FUNCTION_BLOCK FB_DynamicMatrix_Test EXTENDS FB_TestSuite
VAR_INPUT
END_VAR
VAR_OUTPUT
END_VAR
VAR
END_VAR

WhenDeclaredExpectNoMemoryAllocated();
WhenInitiallyResizedExpectMemoryAllocated();
WhenResizedBiggerExpectMoreMemoryAllocated();
WhenResizedSmallerExpectLessMemoryAllocated();
WhenResizedToZeroExpectNoMemoryAllocated();

METHOD PRIVATE WhenDeclaredExpectNoMemoryAllocated
VAR_INPUT
END_VAR
VAR
	M : DynamicMatrix;
	
	ExpectedBufferSize : ULINT := 0;
	ExpectedBufferCount : ULINT := 0;
	
	ActualBufferSize : ULINT;
	ActualBufferCount : ULINT;
END_VAR
TEST('WhenDeclaredExpectNoMemoryAllocated');

// @TEST-RUN
ActualBufferSize := M.MemManager.nAllocatedSize;
ActualBufferCount := M.MemManager.nBufferCount;

// @TEST-ASSERT
AssertEquals(Expected := ExpectedBufferSize,
	Actual := ActualBufferSize,
	Message := 'Matrix buffer size not correct');
AssertEquals(Expected := ExpectedBufferCount,
	Actual := ActualBufferCount,
	Message := 'Matrix buffer count not correct');
	
TEST_FINISHED();
END_METHOD

METHOD PRIVATE WhenInitiallyResizedExpectMemoryAllocated
VAR_INPUT
END_VAR

VAR
	M : DynamicMatrix;
	ResizeSuccess : BOOL;
	
	ExpectedBufferSize : ULINT := 1*SIZEOF(LREAL) + SIZEOF(ULINT);
	ExpectedBufferCount : ULINT := 1;
	
	ActualBufferSize : ULINT;
	ActualBufferCount : ULINT;
END_VAR
TEST('WhenInitiallyResizedExpectMemoryAllocated');

// @TEST-RUN
ResizeSuccess := M.Resize(1,1,FALSE,TRUE);

ActualBufferSize := M.MemManager.nAllocatedSize;
ActualBufferCount := M.MemManager.nBufferCount;


// @TEST-ASSERT
AssertTrue(Condition :=ResizeSuccess,
	message := 'Error on valid initial resize');
AssertEquals(Expected := ExpectedBufferSize,
	Actual := ActualBufferSize,
	Message := 'Matrix buffer size not correct');
AssertEquals(Expected := ExpectedBufferCount,
	Actual := ActualBufferCount,
	Message := 'Matrix buffer count not correct');
	
TEST_FINISHED();
END_METHOD

METHOD PRIVATE WhenResizedBiggerExpectMoreMemoryAllocated
VAR_INPUT
END_VAR
VAR
	M : DynamicMatrix;
	InitialResizeSuccess : BOOL;
	SecondResizeSuccess : BOOL;
	
	ExpectedBufferSize : ULINT := 4*SIZEOF(LREAL) + SIZEOF(ULINT);
	ExpectedBufferCount : ULINT := 1;
	
	ActualBufferSize : ULINT;
	ActualBufferCount : ULINT;
END_VAR
TEST('WhenResizedBiggerExpectMoreMemoryAllocated');

// @TEST-RUN
InitialResizeSuccess := M.Resize(1,1,FALSE,TRUE);
SecondResizeSuccess := M.Resize(2,2,FALSE,TRUE);

ActualBufferSize := M.MemManager.nAllocatedSize;
ActualBufferCount := M.MemManager.nBufferCount;

// @TEST-ASSERT
AssertTrue(Condition :=InitialResizeSuccess,
	message := 'Error on valid initial resize');
AssertTrue(Condition :=SecondResizeSuccess,
	message := 'Error on valid second resize');
AssertEquals(Expected := ExpectedBufferSize,
	Actual := ActualBufferSize,
	Message := 'Matrix buffer size not correct');
AssertEquals(Expected := ExpectedBufferCount,
	Actual := ActualBufferCount,
	Message := 'Matrix buffer count not correct');
	
TEST_FINISHED();
END_METHOD

METHOD PRIVATE WhenResizedSmallerExpectLessMemoryAllocated
VAR_INPUT
END_VAR
VAR
	M : DynamicMatrix;
	InitialResizeSuccess : BOOL;
	SecondResizeSuccess : BOOL;
	
	ExpectedBufferSize : ULINT := 1*SIZEOF(LREAL) + SIZEOF(ULINT);
	ExpectedBufferCount : ULINT := 1;
	
	ActualBufferSize : ULINT;
	ActualBufferCount : ULINT;
END_VAR
TEST('WhenResizedSmallerExpectLessMemoryAllocated');

// @TEST-RUN
InitialResizeSuccess := M.Resize(2,2,FALSE,TRUE);
SecondResizeSuccess := M.Resize(1,1,FALSE,TRUE);

ActualBufferSize := M.MemManager.nAllocatedSize;
ActualBufferCount := M.MemManager.nBufferCount;

// @TEST-ASSERT
AssertTrue(Condition :=InitialResizeSuccess,
	message := 'Error on valid initial resize');
AssertTrue(Condition :=SecondResizeSuccess,
	message := 'Error on valid second resize');
AssertEquals(Expected := ExpectedBufferSize,
	Actual := ActualBufferSize,
	Message := 'Matrix buffer size not correct');
AssertEquals(Expected := ExpectedBufferCount,
	Actual := ActualBufferCount,
	Message := 'Matrix buffer count not correct');
	
TEST_FINISHED();
END_METHOD

METHOD PRIVATE WhenResizedToZeroExpectNoMemoryAllocated
VAR_INPUT
END_VAR
VAR
	M : DynamicMatrix;
	InitialResizeSuccess : BOOL;
	SecondResizeSuccess : BOOL;
	
	ExpectedBufferSize : ULINT := 0;
	ExpectedBufferCount : ULINT := 0;
	
	ActualBufferSize : ULINT;
	ActualBufferCount : ULINT;
END_VAR
TEST('WhenResizedToZeroExpectNoMemoryAllocated');

// @TEST-RUN
InitialResizeSuccess := M.Resize(1,1,FALSE,TRUE);
SecondResizeSuccess := M.Resize(0,0,FALSE,TRUE);

ActualBufferSize := M.MemManager.nAllocatedSize;
ActualBufferCount := M.MemManager.nBufferCount;

// @TEST-ASSERT
AssertTrue(Condition :=InitialResizeSuccess,
	message := 'Error on valid initial resize');
AssertTrue(Condition :=SecondResizeSuccess,
	message := 'Error on valid second resize');
AssertEquals(Expected := ExpectedBufferSize,
	Actual := ActualBufferSize,
	Message := 'Matrix buffer size not correct');
AssertEquals(Expected := ExpectedBufferCount,
	Actual := ActualBufferCount,
	Message := 'Matrix buffer count not correct');
	
TEST_FINISHED();
END_METHOD

END_FUNCTION_BLOCK

(* stored: Version 1.1.0.1, ProductVersion 3.1.4024.9
   POU FB_DynamicMatrix_Test: Id {54635403-dd01-0e43-181c-428b6dbc359d}, SpecialFunc None
   Folder Resize: Id {bfa23fd9-95bb-0df9-1e4f-a4e0bf87e25f}
   Method WhenDeclaredExpectNoMemoryAllocated: Id {e76f40f2-9e5f-0e70-0e41-efbd9edc0c41}
   Method WhenInitiallyResizedExpectMemoryAllocated: Id {e070b58a-7b2e-00c9-236c-e1d4bd9dab24}
   Method WhenResizedBiggerExpectMoreMemoryAllocated: Id {4c144e27-cde9-06d8-2c10-1905086e448a}
   Method WhenResizedSmallerExpectLessMemoryAllocated: Id {f15ddc13-ce40-0f57-1947-8a0c4169fc8b}
   Method WhenResizedToZeroExpectNoMemoryAllocated: Id {44d4a43d-fd60-056f-2d77-91c9b8831470} *)
